FUNCTION NegateGeneralResult : E_GeneralResult
VAR_INPUT
	result		: E_GeneralResult;
END_VAR
VAR
END_VAR


CASE result OF
	E_GeneralResult.OK:
		NegateGeneralResult := E_GeneralResult.NOK;
	E_GeneralResult.NOK:
		NegateGeneralResult := E_GeneralResult.OK;
	E_GeneralResult._TRUE:
		NegateGeneralResult := E_GeneralResult._FALSE;
	E_GeneralResult._FALSE:
		NegateGeneralResult := E_GeneralResult._TRUE;
	ELSE
		NegateGeneralResult := result;
END_CASE

END_FUNCTION

(* stored: Version 1.1.0.1, ProductVersion 3.1.4024.11
   POU NegateGeneralResult: Id {c982e807-bb92-42a8-95dc-1dbb092fd1e8}, SpecialFunc None *)
